% RSLogix 500 project mais longe que eu fui.RSS, saved by version 7.00.00.19 %
PROJECT "UNTITLED"    % processor: MicroLogix 1200 %

PROGRAM FILES
  LAD 2   22 rungs

DATA FILES
  O0 OUTPUT  7 elements
  I1 INPUT  10 elements
  S2 STATUS  66 elements
  B3 BINARY  1 elements
  T4 TIMER  3 elements
  C5 COUNTER  1 elements
  R6 CONTROL  1 elements
  N7 INTEGER  1 elements
  F8 FLOAT  56 elements

LADDER 2
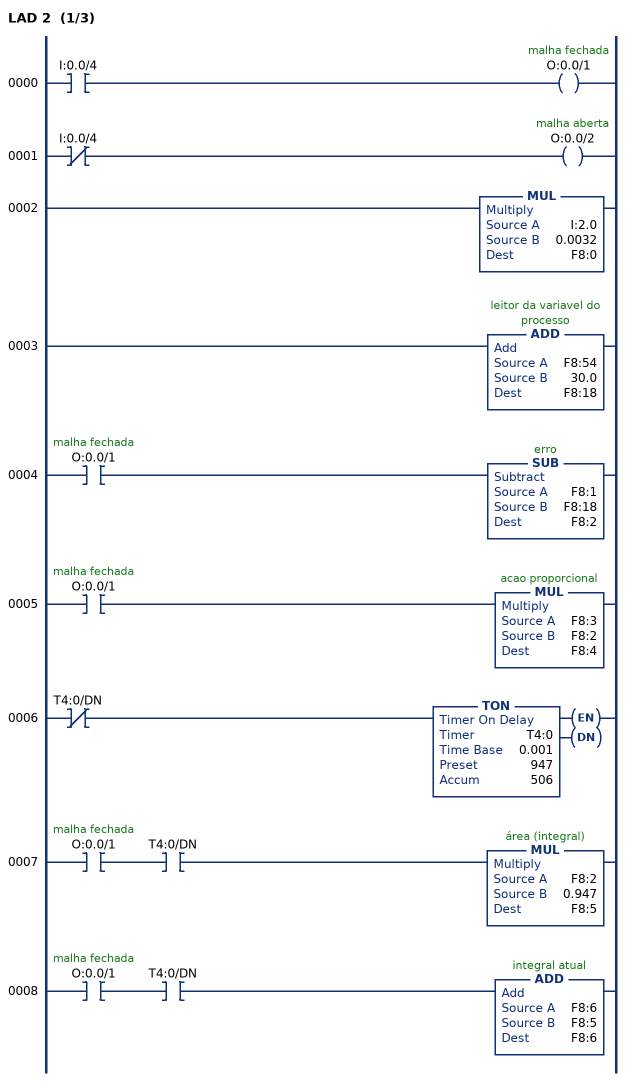
% Rung: 0 %
SOR XIC I:0.0/4 OTE O:0.0/1 EOR
%   O:0.0/1  "malha fechada" %
% Rung: 1 %
SOR XIO I:0.0/4 OTE O:0.0/2 EOR
%   O:0.0/2  "malha aberta" %
% Rung: 2 %
SOR MUL I:2.0 0.0032 F8:0 EOR
% Rung: 3 %
SOR ADD F8:54 30.0 F8:18 EOR
%   F8:18  "leitor da variavel do processo" %
% Rung: 4 %
SOR XIC O:0.0/1 SUB F8:1 F8:18 F8:2 EOR
%   O:0.0/1  "malha fechada" %
%   F8:1  "setpoint" %
%   F8:18  "leitor da variavel do processo" %
%   F8:2  "erro" %
% Rung: 5 %
SOR XIC O:0.0/1 MUL F8:3 F8:2 F8:4 EOR
%   O:0.0/1  "malha fechada" %
%   F8:3  "ganho proporcional" %
%   F8:2  "erro" %
%   F8:4  "acao proporcional" %
% Rung: 6 %
SOR XIO T4:0/DN TON T4:0 0.001 947 506 EOR
% Rung: 7 %
SOR XIC O:0.0/1 XIC T4:0/DN MUL F8:2 0.947 F8:5 EOR
%   O:0.0/1  "malha fechada" %
%   F8:2  "erro" %
%   F8:5  "área (integral)" %
% Rung: 8 %
SOR XIC O:0.0/1 XIC T4:0/DN ADD F8:6 F8:5 F8:6 EOR
%   O:0.0/1  "malha fechada" %
%   F8:6  "integral atual" %
%   F8:5  "área (integral)" %

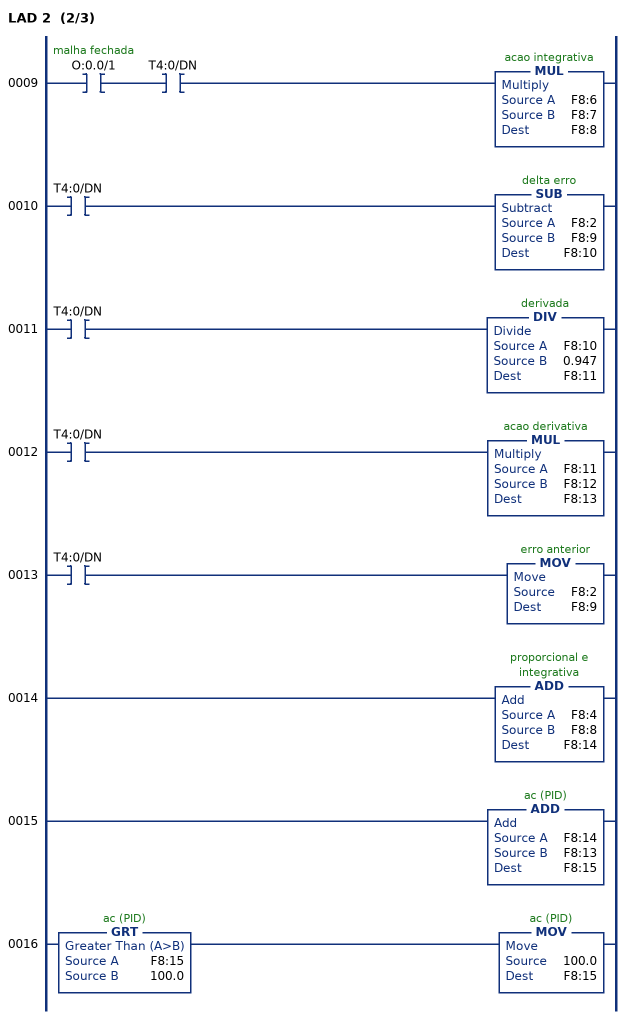
% Rung: 9 %
SOR XIC O:0.0/1 XIC T4:0/DN MUL F8:6 F8:7 F8:8 EOR
%   O:0.0/1  "malha fechada" %
%   F8:6  "integral atual" %
%   F8:7  "ganho integral" %
%   F8:8  "acao integrativa" %
% Rung: 10 %
SOR XIC T4:0/DN SUB F8:2 F8:9 F8:10 EOR
%   F8:2  "erro" %
%   F8:9  "erro anterior" %
%   F8:10  "delta erro" %
% Rung: 11 %
SOR XIC T4:0/DN DIV F8:10 0.947 F8:11 EOR
%   F8:10  "delta erro" %
%   F8:11  "derivada" %
% Rung: 12 %
SOR XIC T4:0/DN MUL F8:11 F8:12 F8:13 EOR
%   F8:11  "derivada" %
%   F8:12  "ganho derivativo" %
%   F8:13  "acao derivativa" %
% Rung: 13 %
SOR XIC T4:0/DN MOV F8:2 F8:9 EOR
%   F8:2  "erro" %
%   F8:9  "erro anterior" %
% Rung: 14 %
SOR ADD F8:4 F8:8 F8:14 EOR
%   F8:4  "acao proporcional" %
%   F8:8  "acao integrativa" %
%   F8:14  "proporcional e integrativa" %
% Rung: 15 %
SOR ADD F8:14 F8:13 F8:15 EOR
%   F8:14  "proporcional e integrativa" %
%   F8:13  "acao derivativa" %
%   F8:15  "ac (PID)" %
% Rung: 16 %
SOR GRT F8:15 100.0 MOV 100.0 F8:15 EOR
%   F8:15  "ac (PID)" %

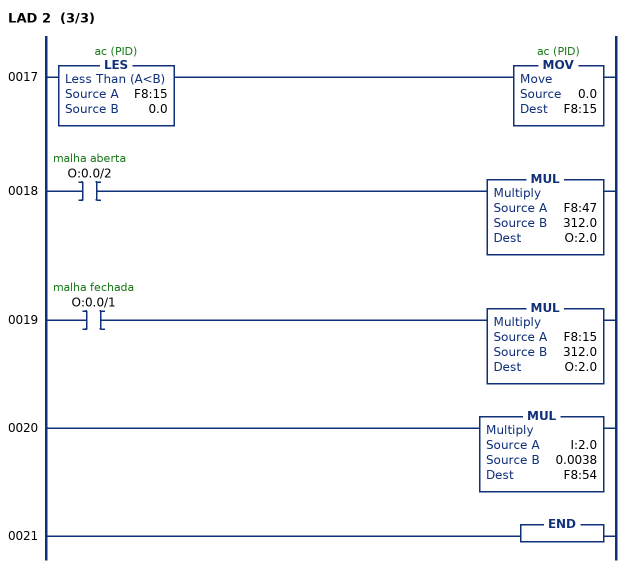
% Rung: 17 %
SOR LES F8:15 0.0 MOV 0.0 F8:15 EOR
%   F8:15  "ac (PID)" %
% Rung: 18 %
SOR XIC O:0.0/2 MUL F8:47 312.0 O:2.0 EOR
%   O:0.0/2  "malha aberta" %
%   F8:47  "acionamento malha aberta" %
% Rung: 19 %
SOR XIC O:0.0/1 MUL F8:15 312.0 O:2.0 EOR
%   O:0.0/1  "malha fechada" %
%   F8:15  "ac (PID)" %
% Rung: 20 %
SOR MUL I:2.0 0.0038 F8:54 EOR
% Rung: 21 %
SOR END EOR

OTHER DOCUMENTED ADDRESSES
  F8:45  "malha fechada"
  F8:46  "malha aberta"
  F8:55  "LEITOR DO VARIAVEL DE PROCESSO"

DATA TABLE (non-zero values as saved)
DATA T4
% .PRE .ACC %
% T4:0 % 947 506
% T4:1 % 244 243
% T4:2 % 1756 716
DATA F8
% F8:0 % 24.2176 50 -8.7584 3.7 -32.40608
% F8:5 % -8.495726 367.4442 0.146 53.64685 -8.971199
% F8:10 % 0.2736015 0.288914 1 0.288914 21.24077
% F8:15 % 21.52969 0 0 58.7584 0
% F8:45 % 0 0 100 0 0
% F8:50 % 0 0 0 0 28.6976
% F8:55 % 32.2496
